TYPE ST_System_AKM_Zustand :
STRUCT
	Betrieb_Anford			: BOOL;
	Betrieb_Soll			: BOOL;
	Betrieb					: BOOL;

	Regelung_Modus			: SINT;
	Regelung_Sollw			: REAL;

	Netze_Anford			: ST_Zustand_Netze_Anford;
	Netz_HW_Anford			: ST_Zustand_Netz_Anford;


	Freigabe				: BOOL;
	Freigabe_Deakt			: BOOL;
	Freigabe_Code			: WORD;

	Stoerung				: BOOL;
	Stoerung_Code			: WORD;

	Warnung					: BOOL;
	Warnung_Code			: WORD;

	Status					: SINT;
	Status_Vorl				: BOOL;
	Status_Nachl			: BOOL;

	Quittierung				: BOOL;

END_STRUCT
END_TYPE

(* stored: Version 1.1.0.1, ProductVersion 3.1.4024.9
   DUT ST_System_AKM_Zustand: Id {aaf326c2-daa2-4f44-ad4c-9882eabcd417} *)
